Staubli VAL3: WriteFile.pgx

program WriteFile(string x_sContent)
begin
  //
  $fileSet(nFileHandle,x_sContent,1)
end
